// TwinCAT 3 PLC project Plc_1
// ProgramVersion: 3.1.4026.23
// libraries:
//   Default, * (Seasight Solutions)
//   Tc2_EtherCAT, * (Beckhoff Automation GmbH)
//   Tc2_Math, * (Beckhoff Automation GmbH)
//   Tc2_Standard, * (Beckhoff Automation GmbH)
//   Tc2_System, * (Beckhoff Automation GmbH)
//   Tc2_Utilities, * (Beckhoff Automation GmbH)
//   Tc3_System_DK, * (Beckhoff - DK)
// project tree:
//   DUTs/ E_ApsState.TcDUT, E_AutoOnOff.TcDUT, E_RmtCmd.TcDUT, E_RmtInCtrl.TcDUT, ST_PitchControl.TcDUT, ST_PitchStatus.TcDUT, ST_RmtLed.TcDUT
//   / FastTask.TcTTO, PlcTask.TcTTO
//   GVLs/ GVL_Constant.TcGVL, GVL_Control.TcGVL, GVL_Gyro.TcGVL, GVL_Persistent.TcGVL, GVL_Misc.TcGVL
//   POUs/ FAST.TcPOU, MAIN.TcPOU
//   POUs/FUNCTION BLOCKS/ FB_Controller.TcPOU, FB_Encoder.TcPOU, FB_DataLogger.TcPOU, FB_Gyro.TcPOU, FB_MovingAverage.TcPOU, FB_PitchMotor.TcPOU, FB_Remote.TcPOU, FB_ThrustMotor.TcPOU
//   POUs/FUNCTIONS/ SystemTimeToString.TcPOU
// real-time tasks:
//   TASK PlcTask: cycle T#1ms, priority 20, ADS port 350
//   TASK FastTask: cycle T#250us, priority 1, ADS port 351
// I/O:
//   DEVICE IO MODULES, AmsNetId 192.168.10.37.3.1
//     K810 (EK1200) [EK1200-5000 EtherCAT Power supply (2A E-Bus)]
//       K811 (EL7031-0030) [EL7031-0030 1Ch. Stepper motor output stage (24V, 2.8A)]
//       K812 (EL7031-0030) [EL7031-0030 1Ch. Stepper motor output stage (24V, 2.8A)]
//       K813 (EL1008) [EL1008 8Ch. Dig. Input 24V, 3ms]
//       K814 (EL2008) [EL2008 8Ch. Dig. Output 24V, 0.5A]
//       K815 (EL1008) [EL1008 8Ch. Dig. Input 24V, 3ms]
//       K816 (EL1008) [EL1008 8Ch. Dig. Input 24V, 3ms]
//       K817 (EL2008) [EL2008 8Ch. Dig. Output 24V, 0.5A]
//       K820 (EL1008) [EL1008 8Ch. Dig. Input 24V, 3ms]
//       K821 (EL1008) [EL1008 8Ch. Dig. Input 24V, 3ms]
//       K822 (EL2008) [EL2008 8Ch. Dig. Output 24V, 0.5A]
//       K823 (EL6224) [EL6224 (IO Link Master)]
//       K824 (EL6070-0033) [EL6070-0033 1Ch. Licence key terminal, individual licences]
//   DEVICE GYRO, AmsNetId 192.168.10.37.4.1
//     Box 15 (EP3751-0260) [EP3751-0260 Acceleration Sensor and Gyroscope]
//   DEVICE VFD 1, AmsNetId 192.168.10.37.6.1
//     Delta MS300 [Delta MS300 EtherCAT(CoE)]
//   DEVICE VFD 2, AmsNetId 192.168.10.37.7.1
//     Delta MS300 [Delta MS300 EtherCAT(CoE)]
// variable links:
//   (this object) <-> GYRO/Box 15 (EP3751-0260)
//     FastTask Inputs/FAST.fbGyro.fGyroTemp <-> AI Sensor Temperature (Real)/Value (Real32)
//     FastTask Inputs/FAST.fbGyro.fGyroVelRawReal <-> AI Gyro Y Samples 1 (Real32)/Samples[0]
//   (this object) <-> IO MODULES/K810 (EK1200)/K811 (EL7031-0030)
//     PlcTask Inputs/MAIN.fbPitchMotor[1].stPitchStat/Error <-> STM Status/Status/Error
//     PlcTask Inputs/MAIN.fbPitchMotor[1].stPitchStat/MovingNegative <-> STM Status/Status/Moving negative
//     PlcTask Inputs/MAIN.fbPitchMotor[1].stPitchStat/MovingPositive <-> STM Status/Status/Moving positive
//     PlcTask Inputs/MAIN.fbPitchMotor[1].stPitchStat/Ready <-> STM Status/Status/Ready
//     PlcTask Inputs/MAIN.fbPitchMotor[1].stPitchStat/ReadyToEnable <-> STM Status/Status/Ready to enable
//     PlcTask Inputs/MAIN.fbPitchMotor[1].stPitchStat/SyncError <-> STM Status/Status/Sync error
//     PlcTask Inputs/MAIN.fbPitchMotor[1].stPitchStat/TorqueReduced <-> STM Status/Status/Torque reduced
//     PlcTask Inputs/MAIN.fbPitchMotor[1].stPitchStat/Warning <-> STM Status/Status/Warning
//     PlcTask Outputs/MAIN.fbPitchMotor[1].stPitchCtrl/Enable <-> STM Control/Control/Enable
//     PlcTask Outputs/MAIN.fbPitchMotor[1].stPitchCtrl/ReduceTorque <-> STM Control/Control/Reduce torque
//     PlcTask Outputs/MAIN.fbPitchMotor[1].stPitchCtrl/Reset <-> STM Control/Control/Reset
//     PlcTask Outputs/MAIN.fbPitchMotor[1].stPitchCtrl/Velocity <-> STM Velocity/Velocity
//   (this object) <-> IO MODULES/K810 (EK1200)/K812 (EL7031-0030)
//     PlcTask Inputs/MAIN.fbPitchMotor[2].stPitchStat/Error <-> STM Status/Status/Error
//     PlcTask Inputs/MAIN.fbPitchMotor[2].stPitchStat/MovingNegative <-> STM Status/Status/Moving negative
//     PlcTask Inputs/MAIN.fbPitchMotor[2].stPitchStat/MovingPositive <-> STM Status/Status/Moving positive
//     PlcTask Inputs/MAIN.fbPitchMotor[2].stPitchStat/Ready <-> STM Status/Status/Ready
//     PlcTask Inputs/MAIN.fbPitchMotor[2].stPitchStat/ReadyToEnable <-> STM Status/Status/Ready to enable
//     PlcTask Inputs/MAIN.fbPitchMotor[2].stPitchStat/SyncError <-> STM Status/Status/Sync error
//     PlcTask Inputs/MAIN.fbPitchMotor[2].stPitchStat/TorqueReduced <-> STM Status/Status/Torque reduced
//     PlcTask Inputs/MAIN.fbPitchMotor[2].stPitchStat/Warning <-> STM Status/Status/Warning
//     PlcTask Outputs/MAIN.fbPitchMotor[2].stPitchCtrl/Enable <-> STM Control/Control/Enable
//     PlcTask Outputs/MAIN.fbPitchMotor[2].stPitchCtrl/ReduceTorque <-> STM Control/Control/Reduce torque
//     PlcTask Outputs/MAIN.fbPitchMotor[2].stPitchCtrl/Reset <-> STM Control/Control/Reset
//     PlcTask Outputs/MAIN.fbPitchMotor[2].stPitchCtrl/Velocity <-> STM Velocity/Velocity
//   (this object) <-> IO MODULES/K810 (EK1200)/K813 (EL1008)
//     PlcTask Inputs/MAIN.b24V1Ok <-> Channel 1/Input
//     PlcTask Inputs/MAIN.b24V2Ok <-> Channel 2/Input
//     PlcTask Inputs/MAIN.fbThrustMotor[1].bPtoSensorOk <-> Channel 3/Input
//     PlcTask Inputs/MAIN.fbThrustMotor[2].bPtoSensorOk <-> Channel 4/Input
//   (this object) <-> IO MODULES/K810 (EK1200)/K814 (EL2008)
//     PlcTask Outputs/MAIN.bGreenLight <-> Channel 1/Output
//     PlcTask Outputs/MAIN.bWarningBuzzer <-> Channel 5/Output
//   (this object) <-> IO MODULES/K810 (EK1200)/K815 (EL1008)
//     PlcTask Inputs/MAIN.fbRemote[1].abRmtBtn[{0..7}] <-> Channel {1..8}/Input  (8 links)
//   (this object) <-> IO MODULES/K810 (EK1200)/K816 (EL1008)
//     PlcTask Inputs/MAIN.fbRemote[1].abRmtBtn[10] <-> Channel 3/Input
//     PlcTask Inputs/MAIN.fbRemote[1].abRmtBtn[8] <-> Channel 1/Input
//     PlcTask Inputs/MAIN.fbRemote[1].abRmtBtn[9] <-> Channel 2/Input
//     PlcTask Inputs/MAIN.fbRemote[1].bOn <-> Channel 8/Input
//     PlcTask Inputs/MAIN.fbRemote[1].bStop <-> Channel 7/Input
//   (this object) <-> IO MODULES/K810 (EK1200)/K817 (EL2008)
//     PlcTask Outputs/MAIN.fbRemote[1].stRmtLed/Alarm <-> Channel 5/Output
//     PlcTask Outputs/MAIN.fbRemote[1].stRmtLed/Hub1 <-> Channel 1/Output
//     PlcTask Outputs/MAIN.fbRemote[1].stRmtLed/Hub2 <-> Channel 4/Output
//     PlcTask Outputs/MAIN.fbRemote[1].stRmtLed/InControl <-> Channel 3/Output
//     PlcTask Outputs/MAIN.fbRemote[1].stRmtLed/On <-> Channel 2/Output
//   (this object) <-> IO MODULES/K810 (EK1200)/K820 (EL1008)
//     PlcTask Inputs/MAIN.fbRemote[2].abRmtBtn[{0..7}] <-> Channel {1..8}/Input  (8 links)
//   (this object) <-> IO MODULES/K810 (EK1200)/K821 (EL1008)
//     PlcTask Inputs/MAIN.fbRemote[2].abRmtBtn[10] <-> Channel 3/Input
//     PlcTask Inputs/MAIN.fbRemote[2].abRmtBtn[8] <-> Channel 1/Input
//     PlcTask Inputs/MAIN.fbRemote[2].abRmtBtn[9] <-> Channel 2/Input
//     PlcTask Inputs/MAIN.fbRemote[2].bOn <-> Channel 8/Input
//     PlcTask Inputs/MAIN.fbRemote[2].bStop <-> Channel 7/Input
//   (this object) <-> IO MODULES/K810 (EK1200)/K822 (EL2008)
//     PlcTask Outputs/MAIN.fbRemote[2].stRmtLed/Alarm <-> Channel 5/Output
//     PlcTask Outputs/MAIN.fbRemote[2].stRmtLed/Hub1 <-> Channel 1/Output
//     PlcTask Outputs/MAIN.fbRemote[2].stRmtLed/Hub2 <-> Channel 4/Output
//     PlcTask Outputs/MAIN.fbRemote[2].stRmtLed/InControl <-> Channel 3/Output
//     PlcTask Outputs/MAIN.fbRemote[2].stRmtLed/On <-> Channel 2/Output
//   (this object) <-> IO MODULES/K810 (EK1200)/K823 (EL6224)
//     PlcTask Inputs/MAIN.fbEncoder[1].bMeasurementValueUnsafe <-> IO-Link Port1/Measurement Value Unsafe
//     PlcTask Inputs/MAIN.fbEncoder[2].bMeasurementValueUnsafe <-> IO-Link Port2/Measurement Value Unsafe
//     PlcTask Inputs/MAIN.fbEncoder[1].bNoMeasurementData <-> IO-Link Port1/Out of Range/No Measurement Data
//     PlcTask Inputs/MAIN.fbEncoder[2].bNoMeasurementData <-> IO-Link Port2/Out of Range/No Measurement Data
//     PlcTask Inputs/MAIN.fbEncoder[1].bOutOfMeasurementRange <-> IO-Link Port1/Out of Measurement Range
//     PlcTask Inputs/MAIN.fbEncoder[2].bOutOfMeasurementRange <-> IO-Link Port2/Out of Measurement Range
//     PlcTask Inputs/MAIN.fbEncoder[1].bSystemError <-> IO-Link Port1/System Error
//     PlcTask Inputs/MAIN.fbEncoder[2].bSystemError <-> IO-Link Port2/System Error
//     PlcTask Inputs/MAIN.fbEncoder[1].nMeasurementValue <-> IO-Link Port1/Measurement Value
//     PlcTask Inputs/MAIN.fbEncoder[2].nMeasurementValue <-> IO-Link Port2/Measurement Value
//     PlcTask Inputs/MAIN.fbEncoder[1].nScalingFactor <-> IO-Link Port1/Scaling Factor
//     PlcTask Inputs/MAIN.fbEncoder[2].nScalingFactor <-> IO-Link Port2/Scaling Factor
//     PlcTask Inputs/MAIN.fbEncoder[1].nStateIo <-> DeviceState Inputs/State Ch1
//     PlcTask Inputs/MAIN.fbEncoder[2].nStateIo <-> DeviceState Inputs/State Ch2
//   (this object) <-> VFD 1/Delta MS300
//     PlcTask Inputs/MAIN.fbThrustMotor[1].fbVfd.nActualCurrent <-> 2nd TxPDO Mapping/[ 2104h ]Output current
//     PlcTask Inputs/MAIN.fbThrustMotor[1].fbVfd.nActualPower <-> 2nd TxPDO Mapping/[ 210Fh ]Power output
//     PlcTask Inputs/MAIN.fbThrustMotor[1].fbVfd.nActualVelocity <-> 2nd TxPDO Mapping/[ 2207h ]motor speed in rpm estimated
//     PlcTask Inputs/MAIN.fbThrustMotor[1].fbVfd.nModeOperationStat <-> 1st TxPDO Mapping/Mode Of Operation Display
//     PlcTask Inputs/MAIN.fbThrustMotor[1].fbVfd.nStatusWord <-> 1st TxPDO Mapping/Status Word
//     PlcTask Outputs/MAIN.fbThrustMotor[1].fbVfd.nControlWord <-> 1st RxPDO Mapping/Control Word
//     PlcTask Outputs/MAIN.fbThrustMotor[1].fbVfd.nModeOperationCtrl <-> 1st RxPDO Mapping/Mode Of Operation
//     PlcTask Outputs/MAIN.fbThrustMotor[1].fbVfd.nRampDownTime <-> 2nd Receive PDO mapping/vl Ramp down time
//     PlcTask Outputs/MAIN.fbThrustMotor[1].fbVfd.nRampUpTime <-> 2nd Receive PDO mapping/vl Ramp up time
//     PlcTask Outputs/MAIN.fbThrustMotor[1].fbVfd.nTargetVelocity <-> 1st RxPDO Mapping/vl target velocity
//   (this object) <-> VFD 2/Delta MS300
//     PlcTask Inputs/MAIN.fbThrustMotor[2].fbVfd.nActualCurrent <-> 2nd TxPDO Mapping/[ 2104h ]Output current
//     PlcTask Inputs/MAIN.fbThrustMotor[2].fbVfd.nActualPower <-> 2nd TxPDO Mapping/[ 210Fh ]Power output
//     PlcTask Inputs/MAIN.fbThrustMotor[2].fbVfd.nActualVelocity <-> 2nd TxPDO Mapping/[ 2207h ]motor speed in rpm estimated
//     PlcTask Inputs/MAIN.fbThrustMotor[2].fbVfd.nModeOperationStat <-> 1st TxPDO Mapping/Mode Of Operation Display
//     PlcTask Inputs/MAIN.fbThrustMotor[2].fbVfd.nStatusWord <-> 1st TxPDO Mapping/Status Word
//     PlcTask Outputs/MAIN.fbThrustMotor[2].fbVfd.nControlWord <-> 1st RxPDO Mapping/Control Word
//     PlcTask Outputs/MAIN.fbThrustMotor[2].fbVfd.nModeOperationCtrl <-> 1st RxPDO Mapping/Mode Of Operation
//     PlcTask Outputs/MAIN.fbThrustMotor[2].fbVfd.nRampDownTime <-> 2nd Receive PDO mapping/vl Ramp down time
//     PlcTask Outputs/MAIN.fbThrustMotor[2].fbVfd.nRampUpTime <-> 2nd Receive PDO mapping/vl Ramp up time
//     PlcTask Outputs/MAIN.fbThrustMotor[2].fbVfd.nTargetVelocity <-> 1st RxPDO Mapping/vl target velocity

CONFIGURATION Plc_1
    RESOURCE PLC ON TwinCAT3
        TASK FastTask(INTERVAL := T#250us, PRIORITY := 1);
        TASK PlcTask(INTERVAL := T#1ms, PRIORITY := 20);
        PROGRAM FAST WITH FastTask : FAST;
        PROGRAM MAIN WITH PlcTask : MAIN;
    END_RESOURCE
END_CONFIGURATION

// ---- DUTs/E_ApsState.TcDUT
{attribute 'qualified_only'}
{attribute 'strict'}
{attribute 'to_string'}
TYPE E_ApsState :
(
	None := 0,
	Off,
	Manual,
	Auto
);
END_TYPE

// ---- DUTs/E_AutoOnOff.TcDUT

{attribute 'to_string'}
TYPE E_AutoOnOff :
(
	Off := 0,
	On
);
END_TYPE

// ---- DUTs/E_RmtCmd.TcDUT
{attribute 'to_string'}
TYPE E_RmtCmd :
(
	None := 0,
	Ccw := 1,
// 	ON := 2,
	Cw := 4,
	RequestControl := 5, // Ccw + Cw
// 	Hub1 := 8,
	StartHub1 := 10, // Hub1 + On
	Off := 16, // Used for Estop
	ResetEstop := 18, // On + Off for 2 seconds
	StopHub1 := 24, // Hub1 + Off
// 	Hub2 := 32,
	StartHub2 := 34, // Hub2 + On
	AutoOnOff := 40, // Hub1 + Hub2
	StopHub2 := 48 // Hub2 + Off
// 	L2B1 := 64,
// 	L2B2 := 128,
// 	L2B3 := 256,
// 	L2B4 := 512,
// 	L2B5 := 1024
);
END_TYPE

// ---- DUTs/E_RmtInCtrl.TcDUT
{attribute 'to_string'}
TYPE E_RmtInCtrl :
(
	None := 0,
	Remote1,
	Remote2
);
END_TYPE

// ---- DUTs/ST_PitchControl.TcDUT
TYPE ST_PitchControl :
STRUCT
	Enable: BOOL;
	Reset: BOOL;
	ReduceTorque: BOOL;
	Velocity: INT;
END_STRUCT
END_TYPE

// ---- DUTs/ST_PitchStatus.TcDUT
TYPE ST_PitchStatus :
STRUCT
	ReadyToEnable: BOOL;
	Ready: BOOL;
	Warning: BOOL;
	Error: BOOL;
	MovingPositive: BOOL;
	MovingNegative: BOOL;
	TorqueReduced: BOOL;
	SyncError: BOOL;
END_STRUCT
END_TYPE

// ---- DUTs/ST_RmtLed.TcDUT
TYPE ST_RmtLed :
STRUCT
	On: BOOL;
	InControl: BOOL;
	Hub1: BOOL;
	Hub2: BOOL;
	Alarm: BOOL;
END_STRUCT
END_TYPE

// ---- GVLs/GVL_Constant.TcGVL
{attribute 'qualified_only'}
VAR_GLOBAL CONSTANT
	fPITCH_LIMIT: LREAL := 10.8; // [deg]
END_VAR

// ---- GVLs/GVL_Control.TcGVL
{attribute 'qualified_only'}
VAR_GLOBAL
	bCalibrateGyro: BOOL := FALSE;
	bResetGryo: BOOL := FALSE;
END_VAR

// ---- GVLs/GVL_Gyro.TcGVL
{attribute 'qualified_only'}
VAR_GLOBAL
	fGyroVel: LREAL;
	fGyroPos: LREAL;
	fGyroPosHmi: LREAL;
	fSetPoint: LREAL;
END_VAR

// ---- GVLs/GVL_Persistent.TcGVL
{attribute 'qualified_only'}
VAR_GLOBAL PERSISTENT
	fOffset: LREAL := 0.0;
	fGyroTempCali: REAL := 0.0;
END_VAR

// ---- GVLs/GVL_Misc.TcGVL
{attribute 'qualified_only'}
VAR_GLOBAL
	eApsState: E_ApsState;
	fPitchTargetPos: LREAL;
END_VAR

// ---- POUs/FAST.TcPOU
PROGRAM FAST
VAR
    fbGyro : FB_Gyro;
    rtCalReq : R_TRIG;
    rtResetReq : R_TRIG;

    bCalPulse : BOOL;
    bResetPulse : BOOL;
	
	fbController: FB_Controller;
	
	eRmtInCtrl: E_RmtInCtrl;
	_eRmtCmd: E_RmtCmd;
END_VAR

// Only receiving Commands form Remote In Control
IF Main.eRmtInCtrl = MAIN.fbRemote[1].eId THEN
	_eRmtCmd := MAIN.fbRemote[1].eRmtCmd;
ELSIF Main.eRmtInCtrl = MAIN.fbRemote[2].eId THEN
	_eRmtCmd := MAIN.fbRemote[2].eRmtCmd;
ELSE
	_eRmtCmd := E_RmtCmd.None;
END_IF


rtCalReq(CLK := GVL_Control.bCalibrateGyro);
rtResetReq(CLK := GVL_Control.bResetGryo);

bCalPulse := rtCalReq.Q;
bResetPulse := rtResetReq.Q;

// optional: clear level requests after edge captured
IF rtCalReq.Q THEN
    GVL_Control.bResetGryo := FALSE;
END_IF
IF rtResetReq.Q THEN
    GVL_Control.bResetGryo := FALSE;
END_IF

fbGyro(
    bCalibrateGyro := bCalPulse,
    bResetGyro := bResetPulse,
    fGyroVel => fbController.fGyroVel,
    fGyroPos => fbController.fGyroPos
);

fbController(
	bStart := (GVL_Misc.eApsState = E_ApsState.Auto),
	bMovSpCw := _eRmtCmd = E_RmtCmd.Cw,
	bMovSpCcw := _eRmtCmd = E_RmtCmd.Ccw,
	fPitchLimit := GVL_Constant.fPITCH_LIMIT,
	fTargetPosition => GVL_Misc.fPitchTargetPos
	);

END_PROGRAM

// ---- POUs/FUNCTION BLOCKS/FB_Gyro.TcPOU
FUNCTION_BLOCK FB_Gyro
VAR_INPUT
    bCalibrateGyro : BOOL;
    bResetGyro : BOOL;
END_VAR
VAR_OUTPUT
    fGyroVel : LREAL;
    fGyroPos : LREAL;
END_VAR
VAR
    bStartTimer : BOOL;
    bInitDone : BOOL;
    bInitFilter : BOOL;

    rtCalibrateGyro : R_TRIG;
    rtResetGyro : R_TRIG;
    rtPersist : R_TRIG;

    tonCalibrateGyro : TON := (PT := tCALIBRATE_GYRO);

    fGyroVelRawReal AT %I* : REAL;
	fGyroTemp AT %I* : REAL;
    fGyroVelRaw : LREAL;
    fOffset : LREAL;

    fSampleHateHz : LREAL := 4000.0;
    fCutoffHz : LREAL := 5.0;

    fbMovAvg : FB_MovingAverage;
    fbWritePersistentData : WritePersistentData;

    nTaskInfo : DINT;
    fCycleTime : LREAL;
	nCnt: INT := 1;
	fGyroTempCali: REAL;
	fAlpha: LREAL;
	fGyroTempFilt: LREAL;
END_VAR
VAR CONSTANT
    tCALIBRATE_GYRO : TIME := T#3M;
END_VAR

IF NOT bInitDone THEN
	fGyroTempCali := GVL_Persistent.fGyroTempCali;
	fbMovAvg(bInit := TRUE, fOffsetInit := GVL_Persistent.fOffset);
    bInitDone := TRUE;
END_IF

nTaskInfo := GETCURTASKINDEXEX();
fCycleTime := TO_LREAL(_TaskInfo[nTaskInfo].CycleTime) / 1.0E07;

fGyroVelRaw := TO_LREAL(fGyroVelRawReal);

rtCalibrateGyro(CLK := bCalibrateGyro);
IF rtCalibrateGyro.Q THEN
    bStartTimer := TRUE;
END_IF

tonCalibrateGyro(IN := bStartTimer);
fbMovAvg(
    bStart := (bStartTimer AND NOT tonCalibrateGyro.Q),
	bInit := FALSE,
    fGyroVelRaw := fGyroVelRaw,
    fOffset => fOffset
);

IF bStartTimer THEN
	fGyroTempCali := fGyroTemp;
END_IF

IF tonCalibrateGyro.Q THEN
    bStartTimer := FALSE;
    bInitFilter := TRUE;
	GVL_Control.bCalibrateGyro := FALSE;
	GVL_Control.bResetGryo := TRUE;
END_IF

// Temperatur Filter
fAlpha := 0.00001;
fGyroTempFilt := fGyroTempFilt + fAlpha * (fGyroTemp - fGyroTempFilt);

// Gyro Velocity med Temperatur kompensation
fGyroVel := fGyroVelRaw - fOffset - (0.033 * (fGyroTempFilt - fGyroTempCali));
// Test sample hver 100ms
IF nCnt >= 40 THEN
	fGyroPos := fGyroPos + fGyroVel * fCycleTime * 40;
	nCnt := 1;
ELSE
	nCnt := nCnt + 1;
END_IF

rtResetGyro(CLK := bResetGyro);
IF rtResetGyro.Q THEN
    fGyroPos := 0.0;
END_IF

rtPersist(CLK := tonCalibrateGyro.Q);
IF rtPersist.Q THEN
    GVL_Persistent.fOffset := fOffset;
	GVL_Persistent.fGyroTempCali := fGyroTempCali;
END_IF

fbWritePersistentData(
    NETID := '',
    PORT := 851,
    START := rtPersist.Q,
    BUSY => ,
    ERR => ,
    ERRID =>
);

GVL_Gyro.fGyroPos := fGyroPos;
GVL_Gyro.fGyroVel := fGyroVel;
GVL_Gyro.fGyroPosHmi := LMOD(fGyroPos, 360.0);
IF GVL_Gyro.fGyroPosHmi < 0.0 THEN GVL_Gyro.fGyroPosHmi := 360.0 + GVL_Gyro.fGyroPosHmi; END_IF

END_FUNCTION_BLOCK

// ---- POUs/FUNCTION BLOCKS/FB_MovingAverage.TcPOU
FUNCTION_BLOCK FB_MovingAverage
VAR_INPUT
	bInit: BOOL;
	bStart: BOOL;
	fGyroVelRaw: LREAL;
	fOffsetInit: LREAL;
END_VAR
VAR_OUTPUT
	fOffset: LREAL;
END_VAR
VAR
	ftStart: F_TRIG;
	fCnt: LREAL;

	fTempOffset: LREAL;
END_VAR

ftStart(CLK := bStart);

IF bStart THEN
	fOffset := 0.0;
	fTempOffset := (fTempOffset * fCnt + fGyroVelRaw) / (fCnt + 1.0);		
	fCnt := fCnt + 1.0;
ELSIF ftStart.Q THEN
	fOffset := fTempOffset;
	fTempOffset := 0.0;	
	fCnt := 0;
END_IF
IF bInit THEN
	fOffset := fOffsetInit;
END_IF

END_FUNCTION_BLOCK

// ---- POUs/FUNCTION BLOCKS/FB_Controller.TcPOU
FUNCTION_BLOCK FB_Controller
VAR_INPUT
	bStart: BOOL;
	bMovSpCcw: BOOL;
	bMovSpCw: BOOL;
	fGyroPos: LREAL;
	fGyroVel: LREAL;
	fPitchLimit: LREAL;
END_VAR
VAR_OUTPUT
	fTargetPosition: LREAL;
END_VAR
VAR
	bActive: BOOL;
	fSetPoint: LREAL;
	rtSetPoint: R_TRIG;
	fError: LREAL;
	fKp: LREAL := 1.2;
	fKi: LREAL := 0.000002;
	fKd: LREAL := 2.4;
	fIntegral: LREAL;
	fPidOutput: LREAL;
	fCycleTime: LREAL := 0.0; // [s]
	nTaskInfo: DINT;
END_VAR
VAR CONSTANT
	fSETPOINT_JOG_VELOCITY: LREAL := 1.0; // [deg/s]
END_VAR

bActive := bStart;
 
nTaskInfo := GETCURTASKINDEXEX();

fCycleTime := TO_LREAL(_TaskInfo[nTaskInfo].CycleTime) / 1.0E7;
 
rtSetPoint(CLK := bActive);

IF rtSetPoint.Q THEN
    fSetPoint := fGyroPos;
    fError := 0.0;
    fIntegral := 0.0;
    fPidOutput := 0.0;
    fTargetPosition := 0.0;
END_IF
 
IF NOT bActive THEN
    fError := 0.0;
    fIntegral := 0.0;
    fPidOutput := 0.0;
    fTargetPosition := 0.0;
ELSE

    IF bMovSpCcw AND NOT bMovSpCw THEN
        fSetPoint := fSetPoint + fSETPOINT_JOG_VELOCITY * fCycleTime;
    ELSIF bMovSpCw AND NOT bMovSpCcw THEN
        fSetPoint := fSetPoint - fSETPOINT_JOG_VELOCITY * fCycleTime;
    END_IF
  	fSetPoint := LIMIT(fGyroPos - 10, fSetPoint, fGyroPos + 10);
  
    fError := fSetPoint - fGyroPos;

    // Kun meget langsom position-retur
    IF ABS(fError) > 0.05 THEN
        fIntegral := fIntegral + fKi * fError * fCycleTime;
    END_IF
 
    fIntegral := LIMIT(-0.2 * fPitchLimit, fIntegral, 0.2 * fPitchLimit);

    // Rate damping er hoveddelen: forsøg at holde gyro-hastighed = 0

    fPidOutput :=
        (fKp * fError)
        + fIntegral
        - (fKd * fGyroVel);
 
    fTargetPosition := LIMIT(-fPitchLimit, fPidOutput, fPitchLimit);
 
    // Anti-windup med D-led inkluderet

    IF fTargetPosition <> fPidOutput THEN
        fIntegral := fTargetPosition - (fKp * fError) + (fKd * fGyroVel);
        fIntegral := LIMIT(-0.2 * fPitchLimit, fIntegral, 0.2 * fPitchLimit);
    END_IF

END_IF

GVL_Gyro.fSetPoint := fSetPoint;

END_FUNCTION_BLOCK

// ---- POUs/MAIN.TcPOU
PROGRAM MAIN
VAR
	sSwVersion: STRING := 'V1.0.0.0'; // digit 1 = main SW version, digit 2 = sub SW version, digit 3 = main HMI version, digit 4 = sub HMI version
	bEstopOk: BOOL;
	
	fPitchTargetPos: LREAL;
	
	fbEncoder: ARRAY[1..2] OF FB_Encoder;
	fbPitchMotor: ARRAY[1..2] OF FB_PitchMotor;
	fbThrustMotor: ARRAY[1..2] OF FB_ThrustMotor;
	fbRemote: ARRAY[1..2] OF FB_Remote;
	
	fbDataLogger: FB_DataLogger;
	
	bHubReady: ARRAY[1..2] OF BOOL;
	bStartHub: ARRAY[1..2] OF BOOL;

	eRmtInCtrl: E_RmtInCtrl;
	eAutoOnOff: E_AutoOnOff;
	
	nIdx: INT;
	
	_eRmtCmd: E_RmtCmd;
	
	b24V1Ok AT %I*: BOOL;
	b24V2Ok AT %I*: BOOL;
	
	bGreenLight AT %Q*: BOOL;
	bWarningBuzzer AT %Q*: BOOL;
	fRefPos: LREAL;
	
	fGyroVel AT %I*: LREAL;
	fGyroPos AT %I*: LREAL;
	
	tonWarningBuzzer: TON := (PT := tWARNING_BUZZER);
	tonStartupHub1: TON := (PT := tSTARTUP_HUB);
	tonStartupHub2: TON := (PT := tSTARTUP_HUB);
	tonInitialization: TON := (PT := tINITIALIZATION);
	rtrigAutoOnOff: R_TRIG;
END_VAR
VAR CONSTANT
	tWARNING_BUZZER: TIME := T#5S;
	tSTARTUP_HUB: TIME := T#1S;
	tINITIALIZATION: TIME := T#20S;
	tAUTO_ON_OFF: TIME := T#1MS;
END_VAR

// ---------------------------------------------------------
// 1. Update remotes first
// ---------------------------------------------------------
FOR nIdx := 1 TO 2 DO
    fbRemote[nIdx](
        bEstopOk := bEstopOk,
        eRmtInCtrl := eRmtInCtrl,
        eId := nIdx,
        bHub1Running := fbThrustMotor[1].stVfdOut.Running,
        bHub2Running := fbThrustMotor[2].stVfdOut.Running,
        bSomethingFailed := NOT (bHubReady[1] AND bHubReady[2] AND b24V1Ok AND b24V2Ok)
    );
END_FOR


// ---------------------------------------------------------
// 2. Only receive commands from Remote In Control
// ---------------------------------------------------------
IF eRmtInCtrl = fbRemote[1].eId THEN
    _eRmtCmd := fbRemote[1].eRmtCmd;
ELSIF eRmtInCtrl = fbRemote[2].eId THEN
    _eRmtCmd := fbRemote[2].eRmtCmd;
ELSE
    _eRmtCmd := E_RmtCmd.None;
END_IF


// ---------------------------------------------------------
// 3. Complete stop - stop both hubs
// ---------------------------------------------------------
IF fbRemote[1].bStopAllHubs OR fbRemote[2].bStopAllHubs THEN
    bStartHub[1] := FALSE;
    bStartHub[2] := FALSE;
    _eRmtCmd := E_RmtCmd.None;
END_IF


// ---------------------------------------------------------
// 4. APS state machine - only once
// ---------------------------------------------------------
A_ApsStateMachine();


// Safety: force stop again after state machine
IF fbRemote[1].bStopAllHubs OR fbRemote[2].bStopAllHubs THEN
    bStartHub[1] := FALSE;
    bStartHub[2] := FALSE;
END_IF


// ---------------------------------------------------------
// 5. Initialization check
// ---------------------------------------------------------
tonInitialization(IN := bEstopOk);

IF NOT (bHubReady[1] OR bHubReady[2]) AND tonInitialization.Q THEN
    bEstopOk := FALSE;
END_IF


// ---------------------------------------------------------
// 6. Audible alarm when the first Hub is started
// ---------------------------------------------------------
tonWarningBuzzer(IN := bWarningBuzzer);

IF tonWarningBuzzer.Q THEN
    bWarningBuzzer := FALSE;
END_IF


// ---------------------------------------------------------
// 7. Startup timeout Hub 1
// ---------------------------------------------------------
tonStartupHub1(IN := bStartHub[1] AND NOT bWarningBuzzer);

IF tonStartupHub1.Q AND NOT fbThrustMotor[1].fbVfd.stOutput.Running THEN
    bStartHub[1] := FALSE;
END_IF


// ---------------------------------------------------------
// 8. Startup timeout Hub 2
// ---------------------------------------------------------
tonStartupHub2(IN := bStartHub[2] AND NOT bWarningBuzzer);

IF tonStartupHub2.Q AND NOT fbThrustMotor[2].fbVfd.stOutput.Running THEN
    bStartHub[2] := FALSE;
END_IF


// ---------------------------------------------------------
// 9. Pitch target position
// Reverse direction of Pitch Motor in hub 1
// ---------------------------------------------------------
fbPitchMotor[1](fTargetPos := -fPitchTargetPos);
fbPitchMotor[2](fTargetPos := fPitchTargetPos);


// ---------------------------------------------------------
// 10. Update hubs
// ---------------------------------------------------------
FOR nIdx := 1 TO 2 DO

    IF fbThrustMotor[nIdx].stVfdOut.Ramping THEN
        fbPitchMotor[nIdx].fTargetPos := 0.0;
    END_IF

    fbEncoder[nIdx]();

    fbPitchMotor[nIdx](
        bEnable := bEstopOk,
        nEncPos := fbEncoder[nIdx].nPosition,
        fPitchLimit := GVL_Constant.fPITCH_LIMIT
    );

    fbThrustMotor[nIdx](
        bEnable := bEstopOk,
        bStart := bStartHub[nIdx] AND NOT bWarningBuzzer
    );

    bHubReady[nIdx] :=
        fbEncoder[nIdx].bReady
        AND fbPitchMotor[nIdx].bReady
        AND fbThrustMotor[nIdx].fbVfd.stOutput.ReadyToRun
        AND NOT fbThrustMotor[nIdx].bBrakeNotReleasedError
        AND NOT fbThrustMotor[nIdx].bPtoSensorError;

    IF NOT bHubReady[nIdx] THEN
        bStartHub[nIdx] := FALSE;
    END_IF

END_FOR


// ---------------------------------------------------------
// 11. Green light
// ---------------------------------------------------------
bGreenLight :=
    bHubReady[1]
    AND bHubReady[2]
    AND b24V1Ok
    AND b24V2Ok;
	
// ---------------------------------------------------------
// 12. Data Logger
// ---------------------------------------------------------
fbDataLogger(bEnableLogging := bEstopOk);

ACTION A_ApsStateMachine:
// APS State is None until bEstopOk = TRUE
IF NOT bEstopOk THEN
	GVL_Misc.eApsState := E_ApsState.None;
ELSIF bEstopOk AND NOT (fbThrustMotor[1].stVfdOut.Running OR fbThrustMotor[2].stVfdOut.Running) THEN
	GVL_Misc.eApsState := E_ApsState.Off;
END_IF



// Switch to Auto On Off
rtrigAutoOnOff(clk := (_eRmtCmd = E_RmtCmd.AutoOnOff));

CASE GVL_Misc.eApsState OF
		
	E_ApsState.Off:		// --- Off --- //
		IF _eRmtCmd = E_RmtCmd.Ccw THEN
			fPitchTargetPos := GVL_Constant.fPITCH_LIMIT;
		ELSIF _eRmtCmd = E_RmtCmd.Cw THEN
			fPitchTargetPos := - GVL_Constant.fPITCH_LIMIT;
		ELSE
			fPitchTargetPos := 0.0;
		END_IF
		
		IF _eRmtCmd = E_RmtCmd.StartHub1 THEN
			bWarningBuzzer := TRUE;
			bStartHub[1] := TRUE;
		END_IF
		
		IF _eRmtCmd = E_RmtCmd.StartHub2 THEN
			bWarningBuzzer := TRUE;
			bStartHub[2] := TRUE;
		END_IF
		
		IF fbThrustMotor[1].stVfdOut.Running OR fbThrustMotor[2].stVfdOut.Running THEN
			GVL_Misc.eApsState := E_ApsState.Manual;
		END_IF
		
	E_ApsState.Manual:	// --- Manual --- //
		// Go to Auto if Remote in Control looses connection
		IF eRmtInCtrl = E_RmtInCtrl.None THEN
			GVL_Misc.eApsState := E_ApsState.Auto;
		END_IF
		
		// Pitching back and forth
		IF _eRmtCmd = E_RmtCmd.Ccw THEN
			fPitchTargetPos := GVL_Constant.fPITCH_LIMIT;
		ELSIF _eRmtCmd = E_RmtCmd.Cw THEN
			fPitchTargetPos := -GVL_Constant.fPITCH_LIMIT;
		ELSE
			fPitchTargetPos := 0.0;
		END_IF
		
		// Starting and stopping the Hubs
		IF _eRmtCmd = E_RmtCmd.StartHub1 THEN
			bStartHub[1] := TRUE;
		ELSIF _eRmtCmd = E_RmtCmd.StartHub2 THEN
			bStartHub[2] := TRUE;
		ELSIF _eRmtCmd = E_RmtCmd.StopHub1 THEN
			bStartHub[1] := FALSE;
		ELSIF _eRmtCmd = E_RmtCmd.StopHub2 THEN
			bStartHub[2] := FALSE;
		END_IF
		
		IF rtrigAutoOnOff.Q THEN
			GVL_Misc.eApsState := E_ApsState.Auto;
			fRefPos := fGyroPos;
			//tonAutoOnOff(IN := FALSE);
		END_IF
		
	E_ApsState.Auto:
	
		fPitchTargetPos := GVL_Misc.fPitchTargetPos;
		// Starting and stopping the Hubs
		IF _eRmtCmd = E_RmtCmd.StartHub1 THEN
			bStartHub[1] := TRUE;
		ELSIF _eRmtCmd = E_RmtCmd.StartHub2 THEN
			bStartHub[2] := TRUE;
		ELSIF _eRmtCmd = E_RmtCmd.StopHub1 THEN
			bStartHub[1] := FALSE;
		ELSIF _eRmtCmd = E_RmtCmd.StopHub2 THEN
			bStartHub[2] := FALSE;
		END_IF
		
		IF rtrigAutoOnOff.Q THEN
			GVL_Misc.eApsState := E_ApsState.Manual;
			//tonAutoOnOff(IN := FALSE);
		END_IF
		
END_CASE
END_ACTION

END_PROGRAM

// ---- POUs/FUNCTION BLOCKS/FB_Encoder.TcPOU
FUNCTION_BLOCK FB_Encoder
VAR_INPUT
END_VAR
VAR_OUTPUT
	bReady: BOOL;
	bError: BOOL;
	nPosition: DINT; // [μm]
END_VAR
VAR
	nStateIo AT %I*: USINT; // 3 means operational, everything else is an error
	nMeasurementValue AT %I*: DINT; // [μm]
	nScalingFactor AT %I*: USINT;
	bMeasurementValueUnsafe AT %I*: BOOL;
	bOutOfMeasurementRange AT %I*: BOOL;
	bNoMeasurementData AT %I*: BOOL;
	bSystemError AT %I*: BOOL;
	
	nFreezeCnt: INT;
	_nPosition: DINT;
END_VAR

nPosition := nMeasurementValue;

bError := nStateIo <> 3 OR bMeasurementValueUnsafe OR bOutOfMeasurementRange OR bNoMeasurementData OR bSystemError;

// Make sure encoder is not frozen at value
IF _nPosition = nPosition THEN 
	nFreezeCnt := nFreezeCnt + 1;
ELSE 
	nFreezeCnt := 0; END_IF
	
IF nFreezeCnt >= 100 THEN bError := TRUE; END_IF

bReady := NOT bError;

_nPosition := nPosition;

END_FUNCTION_BLOCK

// ---- POUs/FUNCTION BLOCKS/FB_PitchMotor.TcPOU
FUNCTION_BLOCK FB_PitchMotor
VAR_INPUT
	bEnable: BOOL;
	bReset: BOOL;
	bReduceTorque: BOOL;

	fTargetPos: LREAL; // [deg]
	nEncPos: DINT; // [μm]
	
	fPitchLimit: LREAL;
END_VAR
VAR_OUTPUT
	bReady: BOOL;
	bError: BOOL;
	
	fActPitchPos: LREAL;
END_VAR
VAR
	stPitchCtrl AT %Q*: ST_PitchControl;
	stPitchStat AT %I*: ST_PitchStatus;
	
	bHomed: BOOL;
	nHomingState: INT;
	tonHoming: TON := (PT := tHOMING);
	
	nPitchingState: INT;
	
	_nEncPos: DINT;
	nCnt: INT;
	
	nEndstopPosition: DINT;
	fMinPos: LREAL;
	fMaxPos: LREAL;
	
	fbDegToUm: FB_LinTrafo;
	fbUmToDeg: FB_LinTrafo;
	
	fTempTargetPos: LREAL;
	nTargetPos: LREAL;
END_VAR
VAR CONSTANT
	tHOMING: TIME := T#10S;
	
	nMAX_VELOCITY: INT := 28800; // [steps/s]
	
	nSTOP_LIMIT: LREAL := 150; // [μm] = [0.15 mm]
	
	nENC_JITTER: DINT := 150; // [μm]
	
	nZERO_TO_MAX_PITCH: DINT := 10400; // [μm]
	
	fPITCH_ARM_LENGTH: REAL := 40000.0; // [μm]T := 
END_VAR

// bEnable will be set to bEstopOk in MAIN
stPitchCtrl.Enable := stPitchStat.ReadyToEnable AND bEnable;

// Reset Output Variables
IF NOT bEnable THEN 
	bReady := FALSE;
	bError := FALSE;
	bHomed := FALSE;
END_IF

// Timer to check if Pitch Motor is stuck
tonHoming(IN := NOT bHomed AND stPitchCtrl.Enable);
IF tonHoming.Q THEN
	stPitchCtrl.Enable := FALSE;
	bError := TRUE;
END_IF

// If Pitch Motor is Enabaled but not Homed
IF NOT bHomed AND stPitchCtrl.Enable THEN	
	A_Homing();
// When Homed the Pitch Motor becomes operational
ELSIF bHomed AND stPitchCtrl.Enable THEN
	bReady := TRUE;
END_IF

// Error and Reset Handling
IF stPitchStat.Error THEN
	stPitchCtrl.Enable := FALSE;
	bError := TRUE;
	bReady := FALSE;
END_IF

stPitchCtrl.Reset := stPitchStat.Error OR bReset;
IF stPitchCtrl.Reset THEN stPitchCtrl.Enable := FALSE; END_IF

// Reduce Torque when Pitch Motor is just holding
IF bReady AND NOT (stPitchStat.MovingPositive OR stPitchStat.MovingNegative) THEN
	stPitchCtrl.ReduceTorque := TRUE;
ELSE
	stPitchCtrl.ReduceTorque := FALSE;
END_IF
fTargetPos := LIMIT(-GVL_Constant.fPITCH_LIMIT, fTargetPos, GVL_Constant.fPITCH_LIMIT);
IF bReady THEN
	// Convert Angle-Degrees to Micro-Meters
	fbDegToUm(
		fInputValue := fTargetPos,
		fInMin := -fPitchLimit,
		fInMax := fPitchLimit,
		fOutMin := fMinPos,
		fOutMax := fMaxPos,
		fOutputValue => fTempTargetPos
		);
	
	// Change Data Type
	nTargetPos := TO_DINT(fTempTargetPos);
	
	// Convert MicroMeters to Angle-Degrees
	fbUmToDeg(
		fInputValue := TO_LREAL(nEncPos),
		fInMin := fMinPos,
		fInMax := fMaxPos,
		fOutMin := -fPitchLimit,
		fOutMax := fPitchLimit,
		fOutputValue => fActPitchPos
		);
	
	// Handlse all movement after Homing is completed
	A_Pitching();
END_IF

ACTION A_Homing:
CASE nHomingState OF
	000:	// Start stepper motor in negative direction
			stPitchCtrl.Velocity := -nMAX_VELOCITY;
			
			// Making sure stepper motor is running
			IF stPitchStat.MovingNegative THEN
				nHomingState := 010;
			END_IF
			
	010:	// Montitor when reaching mechanical endstop
			IF _nEncPos <= nEncPos  AND nEncPos <= 25000 THEN
				nCnt := nCnt + 1;
			ELSE
				nCnt := 0;
			END_IF
			
			IF nCnt >= 10 THEN
				stPitchCtrl.Velocity := 0;
				nCnt := 0;
				nEndstopPosition := nEncPos;
				nHomingState := 020;
			END_IF
			
	020:	// Start stepper motor in positive direction
			stPitchCtrl.Velocity := nMAX_VELOCITY;
			
			// Make sure stepper motor is running
			IF stPitchStat.MovingPositive THEN
				nHomingState := 030;
			END_IF
			
	030:	// Stop stepper motor in center position (Pitch = 0 deg)
			IF nEncPos >= nEndstopPosition + nZERO_TO_MAX_PITCH - nSTOP_LIMIT THEN
				stPitchCtrl.Velocity := 0;
				nHomingState := 000;
				bHomed := TRUE;
				
				// Values used for converting between linear and rotational movement
				fMinPos := TO_REAL(nEndstopPosition + nZERO_TO_MAX_PITCH) - SIN(GVL_Constant.fPITCH_LIMIT * pi / 180.0) * fPITCH_ARM_LENGTH;
				fMaxPos := TO_REAL(nEndstopPosition + nZERO_TO_MAX_PITCH) + SIN(GVL_Constant.fPITCH_LIMIT * pi / 180.0) * fPITCH_ARM_LENGTH;
			END_IF
END_CASE

_nEncPos := nEncPos;
END_ACTION

ACTION A_Pitching:
CASE nPitchingState OF
	000:	// Idle - waiting for pitch command
			stPitchCtrl.Velocity := 0;
			IF nTargetPos < nEncPos - nENC_JITTER THEN
				nPitchingState := 010; // Negative direction
			ELSIF nTargetPos >= nEncPos + nENC_JITTER THEN
				nPitchingState := 020; // Positive direction
			END_IF
			
	010:	// --- MOVING IN NEGATIVE DIRECTION ---
			stPitchCtrl.Velocity := -nMAX_VELOCITY;
			IF stPitchStat.MovingNegative THEN
				nPitchingState := 015;
			END_IF
			
	015:	// --- STOP AT TARGET POSITION ---
			IF nTargetPos >= nEncPos - nSTOP_LIMIT THEN
				stPitchCtrl.Velocity := 0;
				nPitchingState := 000;
			END_IF
			
	020:	// --- MOVING IN POSITIVE DIRECTION ---
			stPitchCtrl.Velocity := nMAX_VELOCITY;
			IF stPitchStat.MovingPositive THEN
				nPitchingState := 025;
			END_IF
			
	025:	// --- STOP AT TARGET POSITION ---
			IF nTargetPos <= nEncPos + nSTOP_LIMIT THEN
				stPitchCtrl.Velocity := 0;
				nPitchingState := 000;
			END_IF
END_CASE
END_ACTION

END_FUNCTION_BLOCK

// ---- POUs/FUNCTION BLOCKS/FB_ThrustMotor.TcPOU
FUNCTION_BLOCK FB_ThrustMotor
VAR_INPUT
	bStart: BOOL;
	bEnable: BOOL;
	
	fRotationSpeed: REAL := 1500; // [rpm]
END_VAR
VAR_OUTPUT
	stVfdOut: ST_Delta_MS300_Output;
	bBrakeNotReleasedError: BOOL;
	bPtoSensorError: BOOL;
END_VAR
VAR
	fbVfd: FB_Delta_MS300;
	bPtoSensorOk AT %I*: BOOL;
	
	tonWaitAfterError: TON := (PT := tWAIT_AFTER_ERROR);
	tonStartupCheck: TON := (PT := tSTARTUP_CHECK);
END_VAR
VAR CONSTANT
	tWAIT_AFTER_ERROR: TIME := T#250MS;
	tSTARTUP_CHECK: TIME := T#2S;
	fMOTOR_CURRENT_NAME_TAG: REAL := 30.7; // [A]
END_VAR

stVfdOut := fbVfd.stOutput;
// Motor parameters
fbVfd.stInput.GearRatio := 1.0;
fbVfd.stInput.RampDownTime := 10.0; // [s]
fbVfd.stInput.RampUpTime := 10.0; // [s]
fbVfd.stInput.Velocity := fRotationSpeed;
fbVfd.stInput.Enable := bEnable;

fbVfd();

// Reset VFD in case of an Error
tonWaitAfterError(IN := NOT fbVfd.stOutput.Fault);
IF fbVfd.stOutput.Fault THEN	
	bStart := FALSE;
	fbVfd.stInput.Reset := TRUE;
ELSE
	fbVfd.stInput.Reset := FALSE;
END_IF

// VFD start conditions
fbVfd.stInput.Start := 	bStart
						AND bPtoSensorOk
						AND tonWaitAfterError.Q
						AND NOT bBrakeNotReleasedError;

// Brake release control
IF fbVfd.stOutput.RampingUp AND fbVfd.stOutput.ActualCurrent > fMOTOR_CURRENT_NAME_TAG * 1.1 THEN
	bBrakeNotReleasedError := TRUE;
ELSE
	bBrakeNotReleasedError := FALSE;
END_IF

bPtoSensorError := NOT bPtoSensorOk;

END_FUNCTION_BLOCK

// ---- POUs/FUNCTION BLOCKS/FB_Remote.TcPOU
FUNCTION_BLOCK FB_Remote
VAR_INPUT
	eId: E_RmtInCtrl;
	
	bHub1Running: BOOL;
	bHub2Running: BOOL;
	
	bSomethingFailed: BOOL;
END_VAR
VAR_OUTPUT
	nBtnSum: INT;
	eRmtCmd: E_RmtCmd;
	bStopAllHubs: BOOL;
END_VAR
VAR_IN_OUT
	bEstopOk: BOOL;
	eRmtInCtrl: E_RmtInCtrl;
END_VAR
VAR
	abRmtBtn AT %I*: ARRAY[0..10] OF BOOL;
	bOn AT %I*: BOOL;
	bStop AT %I*: BOOL;
	stRmtLed AT %Q*: ST_RmtLed;
	rtStop: R_TRIG;
	
	tonResetEstop: TON := (PT := tRESET_ESTOP);
	nIdx: INT;
	
	fbAutoBlink: FB_PulseTrain;
	fbAlarmBlink: FB_PulseTrain;
END_VAR
VAR CONSTANT
	tRESET_ESTOP: TIME := T#2S;
END_VAR

// Decode remote buttons first
A_RmtCmd();

// Blink functions
fbAutoBlink(
    bStart := (GVL_Misc.eApsState = E_ApsState.Auto),
    tPulseOn := T#500MS,
    tPulseOff := T#500MS
);

fbAlarmBlink(bStart := NOT bEstopOk);

// Complete stop - stop both hubs when OFF + STOP are pressed
rtStop(CLK := ((E_RmtCmd.Off = nBtnSum) AND bStop));
bStopAllHubs := rtStop.Q;

// Reset Estop
tonResetEstop(IN := E_RmtCmd.ResetEstop = nBtnSum);
IF tonResetEstop.Q AND NOT bEstopOk THEN
    bEstopOk := TRUE;
    eRmtInCtrl := eId;
END_IF

// Request Control. Can only be done when there is no one in control
IF eRmtInCtrl = E_RmtInCtrl.None AND bEstopOk AND eRmtCmd = E_RmtCmd.RequestControl THEN
    eRmtInCtrl := eId;
END_IF

// Make remote lose Control if it is turned off or Estop is activated
IF (eRmtInCtrl = eId AND NOT bOn) OR NOT bEstopOk THEN
    eRmtInCtrl := E_RmtInCtrl.None;
END_IF

// Update LEDs last
A_RmtLed();

ACTION A_RmtCmd:
nBtnSum := 0;
FOR nIdx := 0 TO 10 DO
	IF abRmtBtn[nIdx] THEN
		nBtnSum := nBtnSum + TO_INT(EXPT(2, nIdx));
	END_IF
END_FOR

CASE nBtnSum OF
	E_RmtCmd.Ccw:
		eRmtCmd := E_RmtCmd.Ccw;
		
	E_RmtCmd.Cw:
		eRmtCmd := E_RmtCmd.Cw;
		
	E_RmtCmd.RequestControl:
		eRmtCmd := E_RmtCmd.RequestControl;
		
	E_RmtCmd.StartHub1:
		eRmtCmd := E_RmtCmd.StartHub1;
		
	E_RmtCmd.ResetEstop:
		eRmtCmd := E_RmtCmd.ResetEstop;
		
	E_RmtCmd.StopHub1:
		eRmtCmd := E_RmtCmd.StopHub1;
		
	E_RmtCmd.StartHub2:
		eRmtCmd := E_RmtCmd.StartHub2;
	
	E_RmtCmd.AutoOnOff:
		eRmtCmd := E_RmtCmd.AutoOnOff;
		
	E_RmtCmd.StopHub2:
		eRmtCmd := E_RmtCmd.StopHub2;
ELSE
	eRmtCmd := E_RmtCmd.None;
END_CASE
END_ACTION

ACTION A_RmtLed:
IF bOn THEN
	stRmtLed.On := TRUE;
END_IF

IF eRmtInCtrl = eId THEN
	stRmtLed.InControl := TRUE;
ELSE
	stRmtLed.InControl := FALSE;
END_IF

IF GVL_Misc.eApsState = E_ApsState.Manual THEN
	IF bHub1Running THEN stRmtLed.Hub1 := TRUE; END_IF
	IF bHub2Running THEN stRmtLed.Hub2 := TRUE; END_IF
END_IF

IF GVL_Misc.eApsState = E_ApsState.Auto THEN
	fbAutoBlink(bStart := GVL_Misc.eApsState = E_ApsState.Auto);
	IF bHub1Running THEN stRmtLed.Hub1 := fbAutoBlink.bPulse; ELSE stRmtLed.Hub1 := FALSE; END_IF
	IF bHub2Running THEN stRmtLed.Hub2 := fbAutoBlink.bPulse; ELSE stRmtLed.Hub2 := FALSE; END_IF	
END_IF

IF NOT bEstopOk THEN
	stRmtLed.Alarm := fbAlarmBlink.bPulse;
ELSIF bEstopOk AND bSomethingFailed THEN
	stRmtLed.Alarm := TRUE;
ELSE
	stRmtLed.Alarm := FALSE;
END_IF

IF NOT bHub1Running THEN stRmtLed.Hub1 := FALSE; END_IF
IF NOT bHub2Running THEN stRmtLed.Hub2 := FALSE; END_IF

IF NOT bOn THEN
	stRmtLed.On := FALSE;
	stRmtLed.InControl := FALSE;
	stRmtLed.Hub1 := FALSE;
	stRmtLed.Hub2 := FALSE;
	stRmtLed.Alarm := FALSE;
	IF eRmtInCtrl = eId THEN
		eRmtInCtrl := E_RmtInCtrl.None;
	END_IF
END_IF
END_ACTION

END_FUNCTION_BLOCK

// ---- POUs/FUNCTION BLOCKS/FB_DataLogger.TcPOU
FUNCTION_BLOCK FB_DataLogger

VAR_INPUT
	bEnableLogging						: BOOL;
END_VAR
VAR
	nState								: USINT;
	
	fbFileOpen							: FB_FileOpen;
	fbFilePuts							: FB_FilePuts;
	fbFileClose							: FB_FileClose;
	
	nCreationTime						: ULINT;
	nNextEntryWrTime					: ULINT;
	nTimeNow							: ULINT;
	sGpString							: STRING(24); // LREAL_TO_FMTSTR messes UP when writting directly to sPtr^. Fucking B...
	sPtr								: POINTER TO T_MaxString;
	nPtr								: POINTER TO USINT;
END_VAR

VAR CONSTANT
	sFILE_PATH							: STRING(30) := '/home/Administrator/datalogs/'; // Set length to n+1 for \0 termination
	sBASE_FILENAME						: STRING(21) := 'APS Datalog '; // Set length to n+1 for \0 termination
	nWRITE_PERIOD						: UDINT := 2500000; // x100 ns
	tFILE_FUN_TOUT						: TIME := T#2S;//:= T#100MS;
END_VAR



CASE nState OF
///////////////////////////////////////////////////////////////////////////////////////////////////////////////////////////////////////
	0: // Include the creation time in the filename and open new file 
///////////////////////////////////////////////////////////////////////////////////////////////////////////////////////////////////////
	IF bEnableLogging THEN
		nCreationTime := F_GetSystemTime() + nWRITE_PERIOD;
		nNextEntryWrTime := nCreationTime;
		fbFileOpen( bExecute := FALSE );
		sPtr := ADR( fbFileOpen.sPathName );
		
		sPtr^ := sFILE_PATH;
		StrPtrToStrEnd( '', sPtr );
		sPtr^ := sBASE_FILENAME;
		StrPtrToStrEnd( '', sPtr );
		SystemTimeToString( sPtr, nCreationTime, TRUE );
		StrPtrToStrEnd( '', sPtr );
		sPtr^ := '.txt';
		
		fbFileOpen(
			nMode := FOPEN_MODEAPPEND OR FOPEN_MODETEXT,
			ePath := PATH_GENERIC,
			tTimeout := tFILE_FUN_TOUT,
			bExecute := TRUE );
		nState := 1;
	END_IF
	
///////////////////////////////////////////////////////////////////////////////////////////////////////////////////////////////////////
	1: // Add header at the first lines in the file
///////////////////////////////////////////////////////////////////////////////////////////////////////////////////////////////////////
	fbFileOpen();
	IF NOT (fbFileOpen.bBusy OR fbFilePuts.bBusy) THEN
		IF fbFileOpen.bError OR NOT bEnableLogging THEN
			nState := 6;
		ELSE
			fbFilePuts( bExecute := FALSE );
			sPtr := ADR( fbFilePuts.sLine );
			
			fbFilePuts(
				hFile := fbFileOpen.hFile,
				tTimeout := tFILE_FUN_TOUT,
				bExecute := TRUE );
			nState := 2;
		END_IF
	END_IF
	
///////////////////////////////////////////////////////////////////////////////////////////////////////////////////////////////////////
	2: // Add line with names of the data fields
///////////////////////////////////////////////////////////////////////////////////////////////////////////////////////////////////////
	fbFilePuts();
	IF NOT fbFilePuts.bBusy THEN
		IF fbFilePuts.bError OR NOT bEnableLogging THEN
			nState := 6;
		ELSE
			fbFilePuts( bExecute := FALSE );
			fbFilePuts.sLine := '$LTime,Hub 1 Power,Hub 2 Power,Hub 1 Current,Hub2 Current,Encoder 1 Pos.,Encoder 2 Pos.,Pos. Ref.,Pos. Est.,Vel. Est.,Remote 1 Cmd,Remote 2 Cmd,APS Mode';
			fbFilePuts( bExecute := TRUE );
			nState := 3;
		END_IF
	END_IF

///////////////////////////////////////////////////////////////////////////////////////////////////////////////////////////////////////
	22: // Add line with names of the data fields
///////////////////////////////////////////////////////////////////////////////////////////////////////////////////////////////////////
	fbFilePuts();
	IF NOT fbFilePuts.bBusy THEN
		IF fbFilePuts.bError OR NOT bEnableLogging THEN
			nState := 6;
		ELSE
			fbFilePuts( bExecute := FALSE );
			fbFilePuts.sLine := ',Operation Mode';
			fbFilePuts( bExecute := TRUE );
			nState := 3;
		END_IF
	END_IF
	
///////////////////////////////////////////////////////////////////////////////////////////////////////////////////////////////////////
	3: // Add line with units of the data fields
///////////////////////////////////////////////////////////////////////////////////////////////////////////////////////////////////////
	fbFilePuts();
	IF NOT fbFilePuts.bBusy THEN
		IF fbFilePuts.bError OR NOT bEnableLogging THEN
			nState := 6;
		ELSE
			fbFilePuts( bExecute := FALSE );
			fbFilePuts.sLine := '$L[-],[kW],[kW],[A],[A],[°],[°],[°],[°],[°/s],[-],[-], [-]';
			fbFilePuts( bExecute := TRUE );
			nState := 4;
		END_IF
	END_IF
	
///////////////////////////////////////////////////////////////////////////////////////////////////////////////////////////////////////
	4: // Finish writing
///////////////////////////////////////////////////////////////////////////////////////////////////////////////////////////////////////
	fbFilePuts();
	IF NOT fbFilePuts.bBusy THEN
		IF fbFilePuts.bError OR NOT bEnableLogging THEN
			nState := 6;
		ELSE
			nState := 5;
		END_IF
	END_IF
	
///////////////////////////////////////////////////////////////////////////////////////////////////////////////////////////////////////
	5: // Add new data entry
///////////////////////////////////////////////////////////////////////////////////////////////////////////////////////////////////////
	IF bEnableLogging THEN
		nTimeNow := F_GetSystemTime();
		IF nTimeNow >= nNextEntryWrTime THEN
		
			nNextEntryWrTime := nNextEntryWrTime + nWRITE_PERIOD;
			fbFilePuts( bExecute := FALSE );
			sPtr := ADR( fbFilePuts.sLine );
			
			fbFilePuts.sLine := '$L';
			SystemTimeToString( ADR(sGpString), nTimeNow, FALSE );
			MEMCPY( sPtr+1, ADR(sGpString)+11, 12 );
			sPtr := sPtr + 13;
			sPtr^ := ',';
			sPtr := sPtr + 1;
			
			sGpString := LREAL_TO_FMTSTR( MAIN.fbThrustMotor[1].stVfdOut.ActualPower, 1, TRUE ); // Root Hub Power
			sPtr^ := sGpString;
			StrPtrToStrEnd( ',', sPtr );
			sGpString := LREAL_TO_FMTSTR( MAIN.fbThrustMotor[2].stVfdOut.ActualPower, 1, TRUE ); // Tip Hub Power
			sPtr^ := sGpString;
			StrPtrToStrEnd( ',', sPtr );
		
			sGpString := LREAL_TO_FMTSTR( MAIN.fbThrustMotor[1].stVfdOut.ActualCurrent, 1, TRUE ); // Root Hub Current
			sPtr^ := sGpString;
			StrPtrToStrEnd( ',', sPtr );
			sGpString := LREAL_TO_FMTSTR( MAIN.fbThrustMotor[2].stVfdOut.ActualCurrent, 1, TRUE ); // Tip Hub Current
			sPtr^ := sGpString;
			StrPtrToStrEnd( ',', sPtr );
			
			sGpString := LREAL_TO_FMTSTR( MAIN.fbPitchMotor[1].fActPitchPos, 0, TRUE ); // Encoder Position
			sPtr^ := sGpString;
			StrPtrToStrEnd( ',', sPtr );
			sGpString := LREAL_TO_FMTSTR( MAIN.fbPitchMotor[2].fActPitchPos, 0, TRUE ); // Encoder Position
			sPtr^ := sGpString;
			StrPtrToStrEnd( ',', sPtr );
			
			sGpString := LREAL_TO_FMTSTR( GVL_Gyro.fSetPoint, 2, TRUE ); // Pos. Ref.
			sPtr^ := sGpString;
			StrPtrToStrEnd( ',', sPtr );
			sGpString := LREAL_TO_FMTSTR( GVL_Gyro.fGyroPos, 2, TRUE ); // Pos. Est.
			sPtr^ := sGpString;
			StrPtrToStrEnd( ',', sPtr );
			
			sGpString := LREAL_TO_FMTSTR( GVL_Gyro.fGyroVel, 2, TRUE ); // Vel. Ref.
			sPtr^ := sGpString;
			StrPtrToStrEnd( ',', sPtr );
			
			sGpString := WORD_TO_STRING( TO_WORD(MAIN.fbRemote[1].nBtnSum) ); // Remote Hub Full
			sPtr^ := sGpString;
			StrPtrToStrEnd( ',', sPtr );
			sGpString := WORD_TO_STRING( TO_WORD(MAIN.fbRemote[2].nBtnSum) ); // Remote Hub Halv
			sPtr^ := sGpString;
			StrPtrToStrEnd( ',', sPtr );


			IF GVL_Misc.eApsState = E_ApsState.Auto THEN
				sGpString := 'Auto'; // Operation Mode
				sPtr^ := sGpString;
			ELSIF GVL_Misc.eApsState = E_ApsState.Manual THEN
				sGpString := 'Manuel'; // Operation Mode
				sPtr^ := sGpString;			
			ELSIF GVL_Misc.eApsState = E_ApsState.Off THEN
				sGpString := 'Off'; // Operation Mode
				sPtr^ := sGpString;					
			END_IF
		
			fbFilePuts( bExecute := TRUE );
			nState := 4;
		END_IF
	ELSE
		nState := 6;
	END_IF
	
///////////////////////////////////////////////////////////////////////////////////////////////////////////////////////////////////////
	6: // Close file
///////////////////////////////////////////////////////////////////////////////////////////////////////////////////////////////////////
	fbFileOpen();
	fbFilePuts();
	fbFileClose();
	IF NOT (fbFileOpen.bBusy OR fbFilePuts.bBusy OR fbFileClose.bBusy) THEN
		fbFileClose( bExecute := FALSE );
		fbFileClose(
			hFile := fbFileOpen.hFile,
			tTimeout := tFILE_FUN_TOUT,
			bExecute := TRUE );
		nState := 7;
	END_IF
	
	7:
	fbFileClose();
	IF NOT fbFileClose.bBusy THEN
		nState := 0;
	END_IF
END_CASE

METHOD PRIVATE StrPtrToStrEnd

VAR_INPUT
	sSep								: STRING(1);
END_VAR

VAR_IN_OUT
	sDst								: POINTER TO STRING;
END_VAR

sDst := sDst + LEN2( sDst );
IF sSep <> '' THEN
	sDst^ := sSep;
	sDst := sDst + 1;
END_IF
END_METHOD

END_FUNCTION_BLOCK

// ---- POUs/FUNCTIONS/SystemTimeToString.TcPOU
FUNCTION SystemTimeToString				: STRING(24) // Set length to n+1 for \0 termination

VAR_INPUT
	sPtr								: POINTER TO STRING;
	nSystemTime							: ULINT;
	bForFilename						: BOOL;
END_VAR

VAR
	tFileTimePtr						: POINTER TO T_FILETIME := ADR(nSystemTime);
	nPtr								: POINTER TO USINT := sPtr;
END_VAR


sPtr^ := SYSTEMTIME_TO_STRING( FILETIME_TO_SYSTEMTIME(tFileTimePtr^) );

// YYYY-MM-DD-hh:mm:ss.xxx
IF bForFilename THEN
	nPtr[10] := 16#5F; // '_'
	nPtr[13] := 16#5F; // '_'
	nPtr[16] := 16#5F; // '_'
	nPtr[19] := 16#5F; // '_'
ELSE
	nPtr[10] := 16#20; // ' '
END_IF

END_FUNCTION
